//{attribute 'qualified_only'}
//{attribute 'strict'}
TYPE E_KBUS_RegisterAccessState : (
	//E_KBUS_IDLE,
	//E_KBUS_REQUEST,
	//E_KBUS_RESPONSE,
	//E_KBUS_READREG,
	//E_KBUS_CHECKDATA,
	//E_KBUS_WRITEREG,
	//E_KBUS_RESETPROCESSDATA,
	//E_KBUS_PROCESSDATA,
	//E_KBUS_DONE
	E_KBUS_DUMMY
);
END_TYPE

(* stored: Version 1.1.0.1
   DUT E_KBUS_RegisterAccessState: Id {e0d2cae8-bf39-4156-99ae-dd5343190738} *)
